# EPICS autosave request: iocBoot/sioc-asta-stats01/pvStats.req
file ../pvStatsCommon.req P=$(P), N=1
file ../pvStatsCommon.req P=$(P), N=2
file ../pvStatsCommon.req P=$(P), N=3
